// SIMATIC S7-200 project (STEP 7-Micro/WIN), CPU 226 REL 02.01

ORGANIZATION_BLOCK MAIN:OB1
TITLE=PROGRAM COMMENTS
BEGIN
Network 1 // Network Title
// Network Comment
LD     Q0.0
O      T41
LD     I0.7
EU
OLD
AN     T37
=      Q0.0
Network 2
LD     Q0.0
TON    T37, 20
Network 3 // Network Title
// Network Comment
LD     Q0.1
O      T37
AN     T38
=      Q0.1
Network 4
LD     Q0.1
TON    T38, 20
Network 5 // Network Title
// Network Comment
LD     Q0.2
O      T38
AN     T39
=      Q0.2
Network 6
LD     Q0.2
TON    T39, 20
Network 7 // Network Title
// Network Comment
LD     Q0.3
O      T39
AN     T40
=      Q0.3
Network 8
LD     Q0.3
TON    T40, 20
Network 9 // Network Title
// Network Comment
LD     Q0.4
O      T40
AN     T41
=      Q0.4
Network 10
LD     Q0.4
TON    T41, 20
END_ORGANIZATION_BLOCK
